// TIA Portal V17 export
// export: Created 2023-12-22T15:03:17.8820718Z, ExportSetting WithDefaults, DisplayName Totally Integrated Automation Portal, DisplayVersion V17, DisplayName TIA Portal Openness, DisplayVersion V17, DisplayName TIA Portal Version Control Interface, DisplayVersion V17, DisplayName STEP 7 Professional, DisplayVersion V17, DisplayName STEP 7 Safety, DisplayVersion V17, DisplayName WinCC Advanced, DisplayVersion V17
DATA_BLOCK "SKV_Logic_DB"   // DB12
VERSION : 0.1
// stored: AutoNumber true, DBAccessibleFromOPCUA true, DBAccessibleFromWebserver true, InstanceOfName SKV_Logic, InstanceOfType FB
"SKV_Logic"
   // VAR RETAIN
   //    Start : Bool;
   //    Start_Up { S7_SetPoint := 'True'} : Bool := FALSE;
   //    Mode : Bool;
   //    "Step" : Int;
   //    LE : Real;
   //    SP : Struct
   //       Max { S7_SetPoint := 'True'} : Real := 0.0;
   //       High { S7_SetPoint := 'True'} : Real := 0.0;
   //       Mid { S7_SetPoint := 'True'} : Real := 0.0;
   //       Low { S7_SetPoint := 'True'} : Real := 0.0;
   //       Min { S7_SetPoint := 'True'} : Real := 0.0;
   //    END_STRUCT;
   // END_VAR
BEGIN
END_DATA_BLOCK
